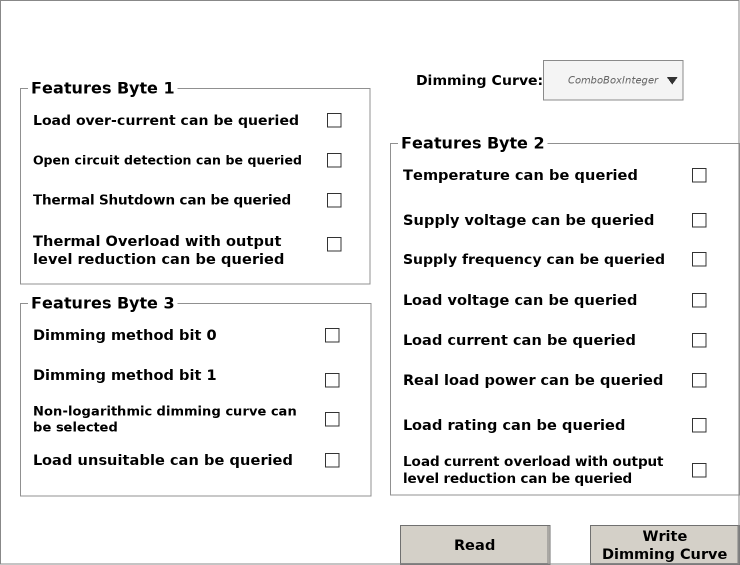
VISUALIZATION Visu_Part205Parameters  // 740x565
    Button (590,525 150x40), "Write Dimming Curve"
        OnMouseClick: execute { DALI_Commissioning.fbPart205Incandescent.bWrite := TRUE; }
    Button (400,525 150x40), "Read"
        OnMouseClick: execute { DALI_Commissioning.fbPart205Incandescent.bReadParameter := TRUE; }
    Group (413,60 270x40)
        Textfield (0,0 130x40), "Dimming Curve:"
        ComboBoxInteger (130,0 140x40), variable: DALI_Commissioning.fbPart205Incandescent.eDimmingCurve, text list: 'DimmingCurve'
    GroupBox (20,80 350x204), "Features Byte 1"
        Textfield (10,25 270x30), "Load over-current can be queried"
        Checkbox (305,25 30x30), variable: DALI_Commissioning.fbPart205Incandescent.bLoadOverCurrentShutdownQueried, input disabled if: True
        Textfield (10,65 270x30), "Open circuit detection can be queried"
        Textfield (10,105 270x30), "Thermal Shutdown can be queried"
        Checkbox (305,65 30x30), variable: DALI_Commissioning.fbPart205Incandescent.bOpenCircuitQueried, input disabled if: true
        Checkbox (305,105 30x30), variable: DALI_Commissioning.fbPart205Incandescent.bThermalShutdownQueried, input disabled if: True
        Textfield (10,150 270x40), "Thermal Overload with output level reduction can be queried"
    GroupBox (390,135 350x360), "Features Byte 2"
        Textfield (10,25 270x30), "Temperature can be queried"
        Checkbox (300,25 30x30), variable: DALI_Commissioning.fbPart205Incandescent.bTempQueried, input disabled if: True
        Textfield (10,65 270x30)
        Textfield (10,65 270x40), "Supply voltage can be queried"
        Textfield (10,150 270x30), "Load voltage can be queried"
        Textfield (10,109 270x30), "Supply frequency can be queried"
        Checkbox (300,70 30x30), variable: DALI_Commissioning.fbPart205Incandescent.bSupplyVoltageQueried, input disabled if: True
        Checkbox (300,150 30x30), variable: DALI_Commissioning.fbPart205Incandescent.bLoadVoltageQueried, input disabled if: True
        Checkbox (300,109 30x30), variable: DALI_Commissioning.fbPart205Incandescent.bSupplyFrequencyQueried, input disabled if: True
        Textfield (10,190 270x30), "Load current can be queried"
        Checkbox (300,190 30x30), variable: DALI_Commissioning.fbPart205Incandescent.bLoadCurrentQueried, input disabled if: True
        Textfield (10,230 270x30), "Real load power can be queried"
        Textfield (10,270 270x40), "Load rating can be queried"
        Textfield (10,320 270x30), "Load current overload with output level reduction can be queried"
        Checkbox (300,230 30x30), variable: DALI_Commissioning.fbPart205Incandescent.bRealLoadPowerQueried, input disabled if: True
        Checkbox (300,275 30x30), variable: DALI_Commissioning.fbPart205Incandescent.bLoadRatingQueried, input disabled if: True
        Checkbox (300,320 30x30), variable: DALI_Commissioning.fbPart205Incandescent.bLoadCurrentOverloadQueried
    GroupBox (20,295 351x201), "Features Byte 3"
        Textfield (10,25 270x30), "Dimming method bit 0"
        Checkbox (303,25 30x30), variable: DALI_Commissioning.fbPart205Incandescent.bDimmingMethodBit0, input disabled if: True
        Textfield (10,65 270x30)
        Textfield (10,65 270x30), "Dimming method bit 1"
        Textfield (10,150 270x30), "Load unsuitable can be queried"
        Textfield (10,109 270x30), "Non-logarithmic dimming curve can be selected"
        Checkbox (303,70 30x30), variable: DALI_Commissioning.fbPart205Incandescent.bDimmingMethodBit1, input disabled if: True
        Checkbox (303,150 30x30), variable: DALI_Commissioning.fbPart205Incandescent.bUnsuitableLoadQueried, input disabled if: True
        Checkbox (303,109 30x30), variable: DALI_Commissioning.fbPart205Incandescent.bNonLogarithmicCurve, input disabled if: True
    Checkbox (325,229 30x30), variable: DALI_Commissioning.fbPart205Incandescent.bThermalOverloadQueried, input disabled if: True
END_VISUALIZATION

(* stored: Version 1.1.0.1, ProductVersion 3.1.4024.12
   Visu Visu_Part205Parameters: Id {f9d1a734-5e4d-4022-b100-637a2ba9112a} *)
